FUNCTION_BLOCK Machine EXTENDS CommonModule IMPLEMENTS I_MachineModule
VAR
	//EMs
	Infeed	: EM_InfeedModule  := (Name := 'Infeed');
	Process : EM_ProcessModule := (Name := 'Process');
	Outfeed : EM_OutfeedModule := (Name := 'Outfeed');

	//Components
	StackLight		 : FB_Component_StackLight		 := (Name := 'StackLight');
	TwinSAFE_Monitor : FB_Component_TwinSAFE_Monitor := (Name := 'TwinSAFE_Monitor');

	//
	fbTON_InfeedRun	   : TON;
	fbTON_ProcessDelay : TON;
	fbTON_OutfeedRun   : TON;

	//
	_CmdMachine : ST_MachineCommand;
	_StsMachine : ST_MachineStatus;
	_RcpMachine : ST_MachineRecipe;
	_CfgMachine : ST_MachineConfig;

	//Visitor
	CollectOEE_MM : FB_CollectOEE;
END_VAR

PROPERTY CfgMachine : REFERENCE TO ST_MachineConfig
GET
CfgMachine REF= _CfgMachine;
END_GET
END_PROPERTY

PROPERTY CmdMachine : REFERENCE TO ST_MachineCommand
GET
CmdMachine REF= _CmdMachine;
END_GET
END_PROPERTY

METHOD CreateCustomModes : BOOL
VAR_INPUT
END_VAR
//Production
CustomModes(eMode						   := E_PMLCustomMode.Production,
			sName						   := 'Production',
			bDisableClearing			   := FALSE,
			bDisableStarting			   := FALSE,
			bDisableSuspended			   := FALSE,
			bDisableStopping			   := FALSE,
			bDisableAborting			   := FALSE,
			bDisableHolding				   := FALSE,
			bDisableHeld				   := FALSE,
			bDisableUnholding			   := FALSE,
			bDisableSuspending			   := FALSE,
			bDisableUnsuspending		   := FALSE,
			bDisableResetting			   := FALSE,
			bDisableIdle				   := FALSE,
			bDisableCompleting			   := FALSE,
			bDisableComplete			   := FALSE,
			bEnableUnitModeChangeStopped   := TRUE,
			bEnableUnitModeChangeIdle	   := TRUE,
			bEnableUnitModeChangeSuspended := TRUE,
			bEnableUnitModeChangeExecute   := TRUE,
			bEnableUnitModeChangeAborted   := TRUE,
			bEnableUnitModeChangeHeld	   := TRUE,
			bEnableUnitModeChangeComplete  := TRUE);

//Home
CustomModes(eMode						   := E_PMLCustomMode.Home,
			sName						   := 'Home',
			bDisableClearing			   := FALSE,
			bDisableStarting			   := FALSE,
			bDisableSuspended			   := FALSE,
			bDisableStopping			   := FALSE,
			bDisableAborting			   := FALSE,
			bDisableHolding				   := FALSE,
			bDisableHeld				   := FALSE,
			bDisableUnholding			   := FALSE,
			bDisableSuspending			   := FALSE,
			bDisableUnsuspending		   := FALSE,
			bDisableResetting			   := FALSE,
			bDisableIdle				   := FALSE,
			bDisableCompleting			   := FALSE,
			bDisableComplete			   := FALSE,
			bEnableUnitModeChangeStopped   := TRUE,
			bEnableUnitModeChangeIdle	   := TRUE,
			bEnableUnitModeChangeSuspended := TRUE,
			bEnableUnitModeChangeExecute   := TRUE,
			bEnableUnitModeChangeAborted   := TRUE,
			bEnableUnitModeChangeHeld	   := TRUE,
			bEnableUnitModeChangeComplete  := TRUE);

//Pre-Positioning for resetting between products
CustomModes(eMode						   := E_PMLCustomMode.PrePositioning,
			sName						   := 'Pre-Positioning',
			bDisableClearing			   := FALSE,
			bDisableStarting			   := FALSE,
			bDisableSuspended			   := FALSE,
			bDisableStopping			   := FALSE,
			bDisableAborting			   := FALSE,
			bDisableHolding				   := FALSE,
			bDisableHeld				   := FALSE,
			bDisableUnholding			   := FALSE,
			bDisableSuspending			   := FALSE,
			bDisableUnsuspending		   := FALSE,
			bDisableResetting			   := FALSE,
			bDisableIdle				   := FALSE,
			bDisableCompleting			   := FALSE,
			bDisableComplete			   := FALSE,
			bEnableUnitModeChangeStopped   := TRUE,
			bEnableUnitModeChangeIdle	   := TRUE,
			bEnableUnitModeChangeSuspended := TRUE,
			bEnableUnitModeChangeExecute   := TRUE,
			bEnableUnitModeChangeAborted   := TRUE,
			bEnableUnitModeChangeHeld	   := TRUE,
			bEnableUnitModeChangeComplete  := TRUE);

//Pre-Production for Heaters
CustomModes(eMode						   := E_PMLCustomMode.PreProduction,
			sName						   := 'Pre-Production',
			bDisableClearing			   := FALSE,
			bDisableStarting			   := FALSE,
			bDisableSuspended			   := FALSE,
			bDisableStopping			   := FALSE,
			bDisableAborting			   := FALSE,
			bDisableHolding				   := FALSE,
			bDisableHeld				   := FALSE,
			bDisableUnholding			   := FALSE,
			bDisableSuspending			   := FALSE,
			bDisableUnsuspending		   := FALSE,
			bDisableResetting			   := FALSE,
			bDisableIdle				   := FALSE,
			bDisableCompleting			   := FALSE,
			bDisableComplete			   := FALSE,
			bEnableUnitModeChangeStopped   := TRUE,
			bEnableUnitModeChangeIdle	   := TRUE,
			bEnableUnitModeChangeSuspended := TRUE,
			bEnableUnitModeChangeExecute   := TRUE,
			bEnableUnitModeChangeAborted   := TRUE,
			bEnableUnitModeChangeHeld	   := TRUE,
			bEnableUnitModeChangeComplete  := TRUE);
END_METHOD

METHOD PUBLIC CyclicLogic
IF NOT _InitComplete THEN
	_InitComplete := Initialize();
	RETURN;
END_IF

//Visitor
Accept(Visitor := CollectOEE_MM);
SUPER^.CyclicLogic();
END_METHOD

//! @summary This method contains code which will execute when this PackML module is in the <b>Execute</b> state
METHOD PROTECTED Execute
(*! <description> <b>The base implementation of this method is empty. User must override this method to provide functionality.</b>
<table> 
	<tr>
		<th> Previous State </th>
		<th> Transition In </th>
		<th> Transition Out </th>
		<th> Next State  </th> 
	</tr>
	<tr>
		<td> Starting<b>-or-</b>Unholding <b>-or-</b>Unsuspending</td>
		<td> State Complete<i>(Starting<b>-or-</b>Unholding<b>-or-</b>Unsuspending)</i></td> 
		<td> State Complete<b>-or-</b>Hold Command<b>-or-</b>Suspend Command</td>
		<td> Completing<b>-or-</b>Holding<b>-or-</b>Suspending</td>
	</tr>
</table>
This method is called as required by <c>StateControl()</c>
</description> 

*)
VAR
END_VAR
CASE _CurrentMode OF
	E_PMLCustomMode.Production:
		CASE DescendantSequenceState OF
			0:
				Infeed.CmdInfeed.StartConveyor := TRUE;
				IF Infeed.StsInfeed.ConveyorRunning THEN
					Infeed.CmdInfeed.StartConveyor := FALSE;
					fbTON_InfeedRun(IN := FALSE);
					DescendantSequenceState := DescendantSequenceState + 10;
				END_IF

			10:
				fbTON_InfeedRun(IN := TRUE, PT := T#3S);
				IF fbTON_InfeedRun.Q THEN
					Infeed.CmdInfeed.StopConveyor := TRUE;
					DescendantSequenceState		  := DescendantSequenceState + 10;
				END_IF

			20:
				IF NOT Infeed.StsInfeed.ConveyorRunning THEN
					Infeed.CmdInfeed.StopConveyor	  := FALSE;
					Process.StsProcess.ProductAtReady := TRUE;
					fbTON_ProcessDelay(IN := FALSE);
					DescendantSequenceState := DescendantSequenceState + 10;
				END_IF

			30:
				fbTON_ProcessDelay(IN := TRUE, PT := T#1.5S);
				IF fbTON_ProcessDelay.Q THEN
					Process.StsProcess.ProductAtReady := FALSE;
					Process.StsProcess.ProductInPos	  := TRUE;
					DescendantSequenceState			  := DescendantSequenceState + 10;
				END_IF

			40:
				IF Process.StsProcess.ProcessComplete THEN
					Process.StsProcess.ProcessComplete := FALSE;
					Outfeed.StsOutfeed.ProductAtReady  := TRUE;
					DescendantSequenceState			   := DescendantSequenceState + 10;
				END_IF

			50:
				IF Outfeed.StsOutfeed.ConveyorRunning THEN
					Outfeed.StsOutfeed.ProductAtReady := FALSE;
					fbTON_OutfeedRun(IN := FALSE);
					DescendantSequenceState := DescendantSequenceState + 10;
				END_IF

			60:
				fbTON_OutfeedRun(IN := TRUE, PT := T#3S);
				IF fbTON_OutfeedRun.Q THEN
					Outfeed.StsOutfeed.ProductRemoved := TRUE;
					DescendantSequenceState			  := DescendantSequenceState + 10;
				END_IF

			70:
				IF NOT Outfeed.StsOutfeed.ConveyorRunning THEN
					Outfeed.StsOutfeed.ProductRemoved := FALSE;
					DescendantSequenceState			  := 0;
				END_IF
		END_CASE

	E_PMLCustomMode.Home:
		_StsCommon.Homed := TRUE;
END_CASE

SUPER^.Execute();
END_METHOD

METHOD PROTECTED Initialize : BOOL
VAR
	i: UDINT;
END_VAR
Initialize := FALSE;
CASE DescendantSequenceState OF
	0: //Register Modules
		RegisterSubmodule(Infeed);
		RegisterSubmodule(Process);
		RegisterSubmodule(Outfeed);

		//Register Components
		RegisterComponent(StackLight);

		//I_CommonModule
		ipCommonModules[1] := Infeed;
		ipCommonModules[2] := Process;
		ipCommonModules[3] := Outfeed;

		//I_CommonComponent
		ipComponents[1] := StackLight;

		//Setup Config
		_LogModeChanges			:= FALSE;
		_LogStateChanges		:= FALSE;
		DescendantSequenceState := DescendantSequenceState + 10;

	10: // Configure Custom Modes
		CreateCustomModes();

		// Copy Mode names
		FOR i := 1 TO 10 DO
			ModeNames[i] := F_UnitModeToString(UDINT_TO_DINT(i));
		END_FOR

		DescendantSequenceState := DescendantSequenceState + 10;

	20:
		//Initialize_Recipes();
		DescendantSequenceState := DescendantSequenceState + 10;

	30: // Call the Super 
		IF SUPER^.Initialize() THEN
			DescendantSequenceState := DescendantSequenceState + 10;
		END_IF

	40:
		Initialize := TRUE;
END_CASE
END_METHOD

PROPERTY RcpMachine : REFERENCE TO ST_MachineRecipe
GET
RcpMachine REF= _RcpMachine;
END_GET
END_PROPERTY

PROPERTY StsMachine : reference to ST_MachineStatus
GET
StsMachine REF= _StsMachine;
END_GET
END_PROPERTY

END_FUNCTION_BLOCK

(* stored: Version 1.1.0.1, ProductVersion 3.1.4024.12
   POU Machine: Id {ae42b527-5b2f-4043-a353-0709b04a7de6}, SpecialFunc None
   Folder Acting: Id {b867810b-83a4-42b8-83fc-d58096ba85df}
   Folder I_CyclicLogic: Id {94db774b-03ec-4ba0-8e48-93f425ae10a5}
   Folder I_MachineModule: Id {c9bacf54-db1c-46d2-bfe4-07954a1811fd}
   Folder Initialize: Id {bd23bc5c-e138-449d-a854-95e1aa4c91d6}
   Folder Waiting: Id {e959f869-19cb-4c34-b909-40dd37320897}
   Property CfgMachine: Id {c2715ec5-865d-4fe1-867b-ae13d7acd5c4}
   Get Get: Id {b93a81a6-d086-45f0-8cb5-2e639d745809}
   Property CmdMachine: Id {d76c054f-aab2-41e6-a61c-f7b4825a5e84}
   Get Get: Id {d8eed551-21f3-4a05-9b2e-18691d2183f7}
   Method CreateCustomModes: Id {d9c82004-48cf-41ac-a536-9c891535f029}
   Method CyclicLogic: Id {f82c43dc-2ed5-48a3-831c-a65c7c1e8bb3}
   Method Execute: Id {756cc64d-9343-460c-b6a2-b999fc29246e}
   Method Initialize: Id {07aaa0ed-cdc4-4c34-8613-f4f8145e0f6a}
   Property RcpMachine: Id {f38b12a8-a6af-4109-ba56-e3b5f1f86775}
   Get Get: Id {d30c764f-8242-4205-a18c-d093f9fe0c82}
   Property StsMachine: Id {3cb6ec70-d991-48b2-a6c4-bc9661147985}
   Get Get: Id {49525a02-5d7a-42f5-8bce-7b90081dab31} *)
